INTERFACE ITF_SPM_OLD

END_INTERFACE

(* stored: Version 1.1.0.1
   Itf ITF_SPM_OLD: Id {9701dffe-a30d-0e0c-0778-f020fa740dc0} *)
